// TIA Portal project "Wine Bottling" (V16)

(* hardware
DEVICE "S71500/ET200MP station_1"  S7-1500 station
   slot 0: "Rail_0"  Rack  6ES7 590-1***0-0AA0
   slot 1: "PLC_1"  CPU 1512C-1 PN  6ES7 512-1CK00-0AB0  V2.8
      slot 3: "CPU display_1"  6ES7591-1AA00-0AA0
      slot 32768: "PROFINET interface_1"  X1
         slot 32769: "Port_1"  X1 P1
         slot 32770: "Port_2"  X1 P2
      slot 34817: "Virtual CP interface port_1"  Virtual CP interface port  Virtual CP interface port
DEVICE "HMI_1"  TP1200 Comfort
   slot 0: "HMI_1"  TP1200 Comfort  6AV2 124-0MC01-0AX0  16.0.0.0
   slot 1: "HMI_RT_1"  TP1200 Comfort  6AV2 124-0MC01-0AX0  16.0.0.0
   slot 5: "HMI_1.IE_CP_1"  PROFINET Interface  16.0.0.0
      slot 1: "PROFINET Interface_1"  PROFINET Interface
         slot 1: "Port_1"  Port
         slot 2: "Port_2"  Port
   slot 7: "HMI_1.MPI/DP_CP_1"  MPI/DP Interface  16.0.0.0
*)

// ===== PLC "PLC_1"  CPU 1512C-1 PN =====

VAR_GLOBAL   // PLC tag table "Default tag table"
   "Start" AT %M0.0 : Bool;
   "Production line" AT %M0.1 : Bool;
   "P_TRIG" AT %M0.2 : Bool;
   "WhiteBottleSensor" AT %M0.3 : Bool;
   "DarkBottleSensor" AT %M0.4 : Bool;
   "Filling" AT %M0.5 : Bool;
   "P_TRIG1" AT %M0.6 : Bool;
   "FillingWhiteWine" AT %M0.7 : Bool;
   "FillingDarkWine" AT %M1.0 : Bool;
   "P_TRIG2" AT %M1.1 : Bool;
   "FilWhite" AT %M1.2 : Bool;
   "FillDark" AT %M1.3 : Bool;
   "P_TRIG3" AT %M1.4 : Bool;
   "P_TRIG4" AT %M1.5 : Bool;
   "P_TRIG5" AT %M1.6 : Bool;
   "Corking" AT %M1.7 : Bool;
   "CorkingWhite" AT %M2.0 : Bool;
   "CorkingDark" AT %M2.1 : Bool;
   "P_TRIG7" AT %M2.2 : Bool;
   "P_TRIG6" AT %M2.3 : Bool;
   "CorkingDarkWine" AT %M2.4 : Bool;
   "P_TRIG8" AT %M2.5 : Bool;
   "CorkingWhiteWine" AT %M2.6 : Bool;
   "P_TRIG9" AT %M2.7 : Bool;
   "P_TRIG10" AT %M3.0 : Bool;
   "Label" AT %M3.1 : Bool;
   "LabelWhite" AT %M3.2 : Bool;
   "LabelDark" AT %M3.3 : Bool;
   "P_TRIG13" AT %M3.4 : Bool;
   "P_TRIG14" AT %M3.5 : Bool;
   "P_TRIG11" AT %M3.6 : Bool;
   "P_TRIG12" AT %M3.7 : Bool;
   "LabelWhiteWine" AT %M4.0 : Bool;
   "LabelDarkWine" AT %M4.1 : Bool;
   "P_TRIG15" AT %M4.2 : Bool;
   "P_TRIG17" AT %M4.3 : Bool;
   "P_TRIG16" AT %M4.4 : Bool;
   "NeckLabeling" AT %M4.5 : Bool;
   "NeckLabelWhite" AT %M4.6 : Bool;
   "NeckLabelDark" AT %M4.7 : Bool;
   "P_TRIG19" AT %M5.0 : Bool;
   "P_TRIG18" AT %M5.1 : Bool;
   "NeckLabelWhiteWine" AT %M5.2 : Bool;
   "NeckLabelDarkWine" AT %M5.3 : Bool;
   "P_TRIG20" AT %M5.4 : Bool;
END_VAR

ORGANIZATION_BLOCK "Main"   // OB1, LAD, ProgramCycle
TITLE = "Main Program Sweep (Cycle)"
{ S7_Optimized_Access := 'TRUE' }
VERSION : 0.1
   VAR_INPUT
      Initial_Call : Bool;   // Initial call of this OB
      Remanence : Bool;   // =True, if remanent data are available
   END_VAR
   VAR_TEMP   // added for the SCL form of the ladder/FBD networks
      _w1 : Bool;
      _w2 : Bool;
      _w3 : Bool;
      _w4 : Bool;
   END_VAR
BEGIN

REGION Network 1
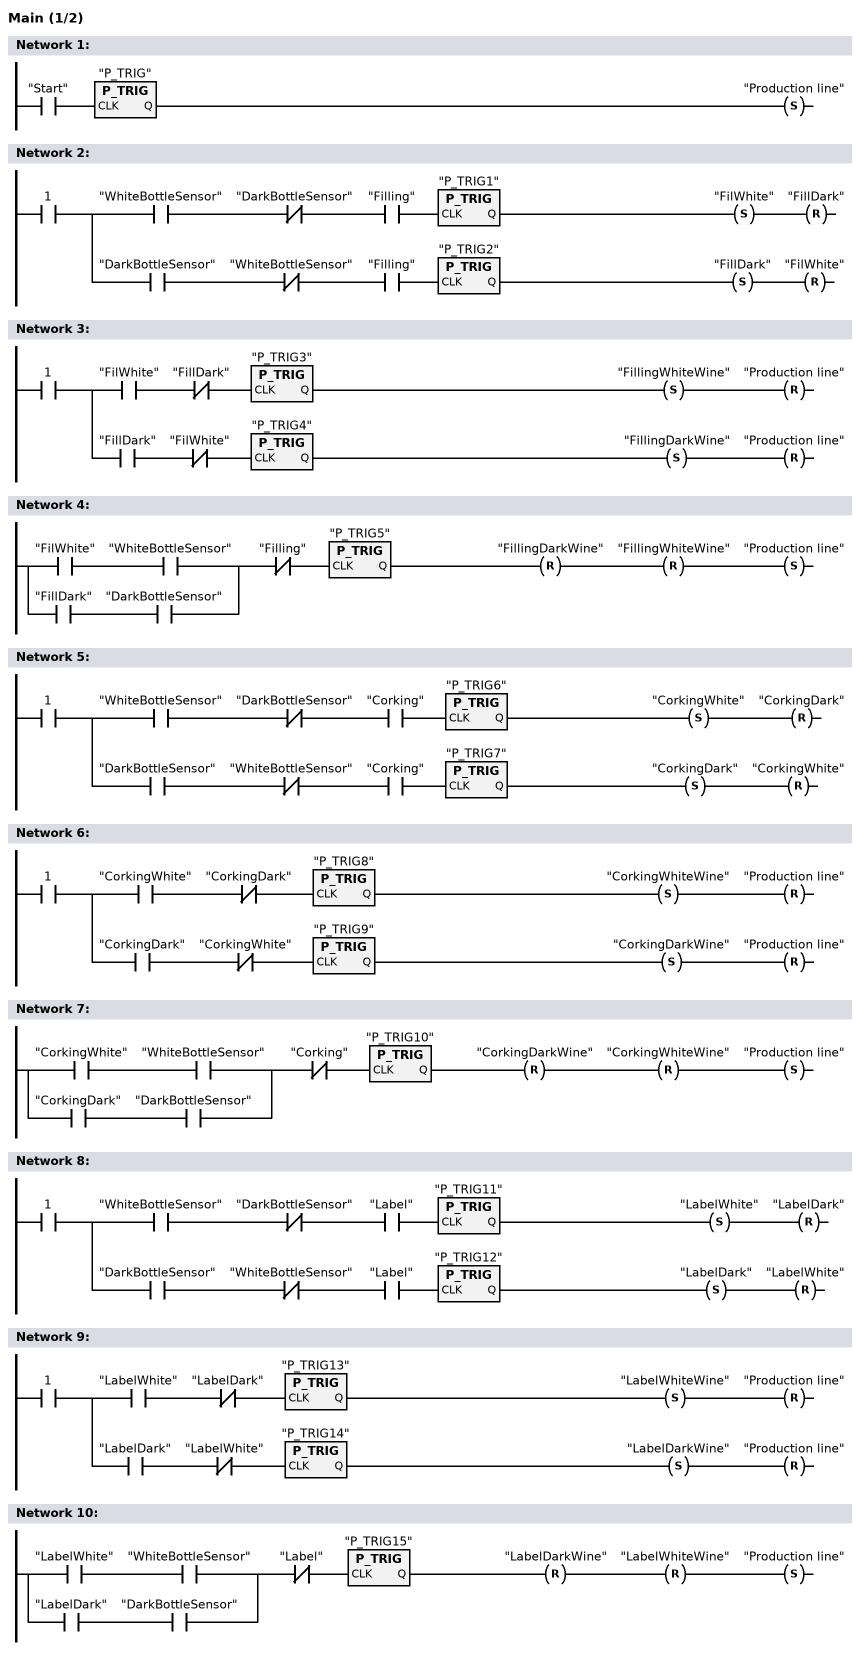
   RUNG wire#powerrail
      Contact( "Start" )
      P_Trig( "P_TRIG" )
      S_Coil( "Production line" )
   END_RUNG
   // the same network as SCL:
   #_w1 := "Start" AND NOT "P_TRIG";   // rising edge
   "P_TRIG" := "Start";
   IF #_w1 THEN "Production line" := TRUE; END_IF;
END_REGION

REGION Network 2
   RUNG wire#powerrail
      Contact( 1 )
      wire#w1
      Contact( "WhiteBottleSensor" )
      I_Contact( "DarkBottleSensor" )
      Contact( "Filling" )
      P_Trig( "P_TRIG1" )
      S_Coil( "FilWhite" )
      R_Coil( "FillDark" )
   END_RUNG
   RUNG wire#w1
      Contact( "DarkBottleSensor" )
      I_Contact( "WhiteBottleSensor" )
      Contact( "Filling" )
      P_Trig( "P_TRIG2" )
      S_Coil( "FillDark" )
      R_Coil( "FilWhite" )
   END_RUNG
   // the same network as SCL:
   #_w1 := 1 AND "WhiteBottleSensor" AND NOT "DarkBottleSensor" AND "Filling";
   #_w2 := #_w1 AND NOT "P_TRIG1";   // rising edge
   "P_TRIG1" := #_w1;
   IF #_w2 THEN
       "FilWhite" := TRUE;
       "FillDark" := FALSE;
   END_IF;
   #_w3 := 1 AND "DarkBottleSensor" AND NOT "WhiteBottleSensor" AND "Filling";
   #_w4 := #_w3 AND NOT "P_TRIG2";   // rising edge
   "P_TRIG2" := #_w3;
   IF #_w4 THEN
       "FillDark" := TRUE;
       "FilWhite" := FALSE;
   END_IF;
END_REGION

REGION Network 3
   RUNG wire#powerrail
      Contact( 1 )
      wire#w1
      Contact( "FilWhite" )
      I_Contact( "FillDark" )
      P_Trig( "P_TRIG3" )
      S_Coil( "FillingWhiteWine" )
      R_Coil( "Production line" )
   END_RUNG
   RUNG wire#w1
      Contact( "FillDark" )
      I_Contact( "FilWhite" )
      P_Trig( "P_TRIG4" )
      S_Coil( "FillingDarkWine" )
      R_Coil( "Production line" )
   END_RUNG
   // the same network as SCL:
   #_w1 := 1 AND "FilWhite" AND NOT "FillDark";
   #_w2 := #_w1 AND NOT "P_TRIG3";   // rising edge
   "P_TRIG3" := #_w1;
   IF #_w2 THEN
       "FillingWhiteWine" := TRUE;
       "Production line" := FALSE;
   END_IF;
   #_w3 := 1 AND "FillDark" AND NOT "FilWhite";
   #_w4 := #_w3 AND NOT "P_TRIG4";   // rising edge
   "P_TRIG4" := #_w3;
   IF #_w4 THEN
       "FillingDarkWine" := TRUE;
       "Production line" := FALSE;
   END_IF;
END_REGION

REGION Network 4
   RUNG wire#powerrail
      Contact( "FilWhite" )
      Contact( "WhiteBottleSensor" )
      wire#w1
      I_Contact( "Filling" )
      P_Trig( "P_TRIG5" )
      R_Coil( "FillingDarkWine" )
      R_Coil( "FillingWhiteWine" )
      S_Coil( "Production line" )
   END_RUNG
   RUNG wire#powerrail
      Contact( "FillDark" )
      Contact( "DarkBottleSensor" )
   END_RUNG wire#w1
   // the same network as SCL:
   #_w1 := (("FilWhite" AND "WhiteBottleSensor") OR ("FillDark" AND "DarkBottleSensor")) AND NOT "Filling";
   #_w2 := #_w1 AND NOT "P_TRIG5";   // rising edge
   "P_TRIG5" := #_w1;
   IF #_w2 THEN
       "FillingDarkWine" := FALSE;
       "FillingWhiteWine" := FALSE;
       "Production line" := TRUE;
   END_IF;
END_REGION

REGION Network 5
   RUNG wire#powerrail
      Contact( 1 )
      wire#w1
      Contact( "WhiteBottleSensor" )
      I_Contact( "DarkBottleSensor" )
      Contact( "Corking" )
      P_Trig( "P_TRIG6" )
      S_Coil( "CorkingWhite" )
      R_Coil( "CorkingDark" )
   END_RUNG
   RUNG wire#w1
      Contact( "DarkBottleSensor" )
      I_Contact( "WhiteBottleSensor" )
      Contact( "Corking" )
      P_Trig( "P_TRIG7" )
      S_Coil( "CorkingDark" )
      R_Coil( "CorkingWhite" )
   END_RUNG
   // the same network as SCL:
   #_w1 := 1 AND "WhiteBottleSensor" AND NOT "DarkBottleSensor" AND "Corking";
   #_w2 := #_w1 AND NOT "P_TRIG6";   // rising edge
   "P_TRIG6" := #_w1;
   IF #_w2 THEN
       "CorkingWhite" := TRUE;
       "CorkingDark" := FALSE;
   END_IF;
   #_w3 := 1 AND "DarkBottleSensor" AND NOT "WhiteBottleSensor" AND "Corking";
   #_w4 := #_w3 AND NOT "P_TRIG7";   // rising edge
   "P_TRIG7" := #_w3;
   IF #_w4 THEN
       "CorkingDark" := TRUE;
       "CorkingWhite" := FALSE;
   END_IF;
END_REGION

REGION Network 6
   RUNG wire#powerrail
      Contact( 1 )
      wire#w1
      Contact( "CorkingWhite" )
      I_Contact( "CorkingDark" )
      P_Trig( "P_TRIG8" )
      S_Coil( "CorkingWhiteWine" )
      R_Coil( "Production line" )
   END_RUNG
   RUNG wire#w1
      Contact( "CorkingDark" )
      I_Contact( "CorkingWhite" )
      P_Trig( "P_TRIG9" )
      S_Coil( "CorkingDarkWine" )
      R_Coil( "Production line" )
   END_RUNG
   // the same network as SCL:
   #_w1 := 1 AND "CorkingWhite" AND NOT "CorkingDark";
   #_w2 := #_w1 AND NOT "P_TRIG8";   // rising edge
   "P_TRIG8" := #_w1;
   IF #_w2 THEN
       "CorkingWhiteWine" := TRUE;
       "Production line" := FALSE;
   END_IF;
   #_w3 := 1 AND "CorkingDark" AND NOT "CorkingWhite";
   #_w4 := #_w3 AND NOT "P_TRIG9";   // rising edge
   "P_TRIG9" := #_w3;
   IF #_w4 THEN
       "CorkingDarkWine" := TRUE;
       "Production line" := FALSE;
   END_IF;
END_REGION

REGION Network 7
   RUNG wire#powerrail
      Contact( "CorkingWhite" )
      Contact( "WhiteBottleSensor" )
      wire#w1
      I_Contact( "Corking" )
      P_Trig( "P_TRIG10" )
      R_Coil( "CorkingDarkWine" )
      R_Coil( "CorkingWhiteWine" )
      S_Coil( "Production line" )
   END_RUNG
   RUNG wire#powerrail
      Contact( "CorkingDark" )
      Contact( "DarkBottleSensor" )
   END_RUNG wire#w1
   // the same network as SCL:
   #_w1 := (("CorkingWhite" AND "WhiteBottleSensor") OR ("CorkingDark" AND "DarkBottleSensor")) AND NOT "Corking";
   #_w2 := #_w1 AND NOT "P_TRIG10";   // rising edge
   "P_TRIG10" := #_w1;
   IF #_w2 THEN
       "CorkingDarkWine" := FALSE;
       "CorkingWhiteWine" := FALSE;
       "Production line" := TRUE;
   END_IF;
END_REGION

REGION Network 8
   RUNG wire#powerrail
      Contact( 1 )
      wire#w1
      Contact( "WhiteBottleSensor" )
      I_Contact( "DarkBottleSensor" )
      Contact( "Label" )
      P_Trig( "P_TRIG11" )
      S_Coil( "LabelWhite" )
      R_Coil( "LabelDark" )
   END_RUNG
   RUNG wire#w1
      Contact( "DarkBottleSensor" )
      I_Contact( "WhiteBottleSensor" )
      Contact( "Label" )
      P_Trig( "P_TRIG12" )
      S_Coil( "LabelDark" )
      R_Coil( "LabelWhite" )
   END_RUNG
   // the same network as SCL:
   #_w1 := 1 AND "WhiteBottleSensor" AND NOT "DarkBottleSensor" AND "Label";
   #_w2 := #_w1 AND NOT "P_TRIG11";   // rising edge
   "P_TRIG11" := #_w1;
   IF #_w2 THEN
       "LabelWhite" := TRUE;
       "LabelDark" := FALSE;
   END_IF;
   #_w3 := 1 AND "DarkBottleSensor" AND NOT "WhiteBottleSensor" AND "Label";
   #_w4 := #_w3 AND NOT "P_TRIG12";   // rising edge
   "P_TRIG12" := #_w3;
   IF #_w4 THEN
       "LabelDark" := TRUE;
       "LabelWhite" := FALSE;
   END_IF;
END_REGION

REGION Network 9
   RUNG wire#powerrail
      Contact( 1 )
      wire#w1
      Contact( "LabelWhite" )
      I_Contact( "LabelDark" )
      P_Trig( "P_TRIG13" )
      S_Coil( "LabelWhiteWine" )
      R_Coil( "Production line" )
   END_RUNG
   RUNG wire#w1
      Contact( "LabelDark" )
      I_Contact( "LabelWhite" )
      P_Trig( "P_TRIG14" )
      S_Coil( "LabelDarkWine" )
      R_Coil( "Production line" )
   END_RUNG
   // the same network as SCL:
   #_w1 := 1 AND "LabelWhite" AND NOT "LabelDark";
   #_w2 := #_w1 AND NOT "P_TRIG13";   // rising edge
   "P_TRIG13" := #_w1;
   IF #_w2 THEN
       "LabelWhiteWine" := TRUE;
       "Production line" := FALSE;
   END_IF;
   #_w3 := 1 AND "LabelDark" AND NOT "LabelWhite";
   #_w4 := #_w3 AND NOT "P_TRIG14";   // rising edge
   "P_TRIG14" := #_w3;
   IF #_w4 THEN
       "LabelDarkWine" := TRUE;
       "Production line" := FALSE;
   END_IF;
END_REGION

REGION Network 10
   RUNG wire#powerrail
      Contact( "LabelWhite" )
      Contact( "WhiteBottleSensor" )
      wire#w1
      I_Contact( "Label" )
      P_Trig( "P_TRIG15" )
      R_Coil( "LabelDarkWine" )
      R_Coil( "LabelWhiteWine" )
      S_Coil( "Production line" )
   END_RUNG
   RUNG wire#powerrail
      Contact( "LabelDark" )
      Contact( "DarkBottleSensor" )
   END_RUNG wire#w1
   // the same network as SCL:
   #_w1 := (("LabelWhite" AND "WhiteBottleSensor") OR ("LabelDark" AND "DarkBottleSensor")) AND NOT "Label";
   #_w2 := #_w1 AND NOT "P_TRIG15";   // rising edge
   "P_TRIG15" := #_w1;
   IF #_w2 THEN
       "LabelDarkWine" := FALSE;
       "LabelWhiteWine" := FALSE;
       "Production line" := TRUE;
   END_IF;
END_REGION

REGION Network 11
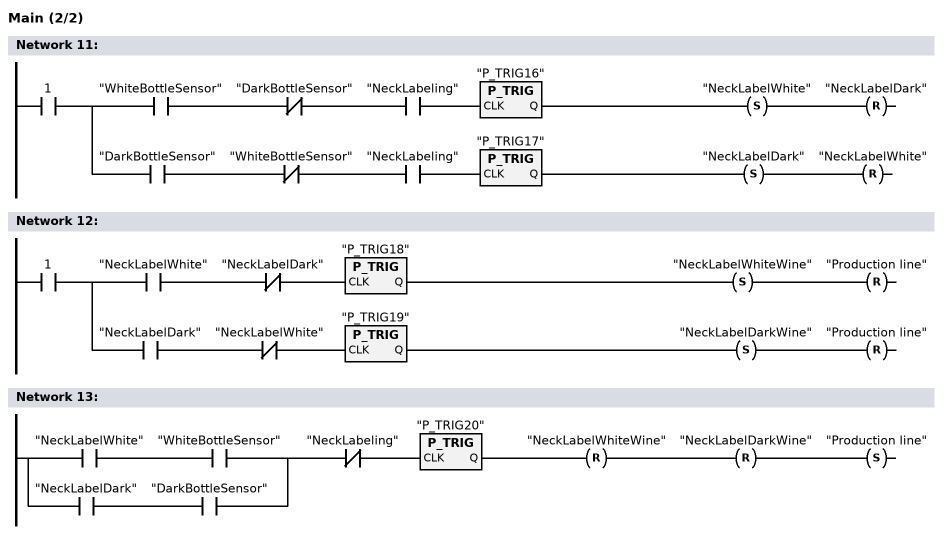
   RUNG wire#powerrail
      Contact( 1 )
      wire#w1
      Contact( "WhiteBottleSensor" )
      I_Contact( "DarkBottleSensor" )
      Contact( "NeckLabeling" )
      P_Trig( "P_TRIG16" )
      S_Coil( "NeckLabelWhite" )
      R_Coil( "NeckLabelDark" )
   END_RUNG
   RUNG wire#w1
      Contact( "DarkBottleSensor" )
      I_Contact( "WhiteBottleSensor" )
      Contact( "NeckLabeling" )
      P_Trig( "P_TRIG17" )
      S_Coil( "NeckLabelDark" )
      R_Coil( "NeckLabelWhite" )
   END_RUNG
   // the same network as SCL:
   #_w1 := 1 AND "WhiteBottleSensor" AND NOT "DarkBottleSensor" AND "NeckLabeling";
   #_w2 := #_w1 AND NOT "P_TRIG16";   // rising edge
   "P_TRIG16" := #_w1;
   IF #_w2 THEN
       "NeckLabelWhite" := TRUE;
       "NeckLabelDark" := FALSE;
   END_IF;
   #_w3 := 1 AND "DarkBottleSensor" AND NOT "WhiteBottleSensor" AND "NeckLabeling";
   #_w4 := #_w3 AND NOT "P_TRIG17";   // rising edge
   "P_TRIG17" := #_w3;
   IF #_w4 THEN
       "NeckLabelDark" := TRUE;
       "NeckLabelWhite" := FALSE;
   END_IF;
END_REGION

REGION Network 12
   RUNG wire#powerrail
      Contact( 1 )
      wire#w1
      Contact( "NeckLabelWhite" )
      I_Contact( "NeckLabelDark" )
      P_Trig( "P_TRIG18" )
      S_Coil( "NeckLabelWhiteWine" )
      R_Coil( "Production line" )
   END_RUNG
   RUNG wire#w1
      Contact( "NeckLabelDark" )
      I_Contact( "NeckLabelWhite" )
      P_Trig( "P_TRIG19" )
      S_Coil( "NeckLabelDarkWine" )
      R_Coil( "Production line" )
   END_RUNG
   // the same network as SCL:
   #_w1 := 1 AND "NeckLabelWhite" AND NOT "NeckLabelDark";
   #_w2 := #_w1 AND NOT "P_TRIG18";   // rising edge
   "P_TRIG18" := #_w1;
   IF #_w2 THEN
       "NeckLabelWhiteWine" := TRUE;
       "Production line" := FALSE;
   END_IF;
   #_w3 := 1 AND "NeckLabelDark" AND NOT "NeckLabelWhite";
   #_w4 := #_w3 AND NOT "P_TRIG19";   // rising edge
   "P_TRIG19" := #_w3;
   IF #_w4 THEN
       "NeckLabelDarkWine" := TRUE;
       "Production line" := FALSE;
   END_IF;
END_REGION

REGION Network 13
   RUNG wire#powerrail
      Contact( "NeckLabelWhite" )
      Contact( "WhiteBottleSensor" )
      wire#w1
      I_Contact( "NeckLabeling" )
      P_Trig( "P_TRIG20" )
      R_Coil( "NeckLabelWhiteWine" )
      R_Coil( "NeckLabelDarkWine" )
      S_Coil( "Production line" )
   END_RUNG
   RUNG wire#powerrail
      Contact( "NeckLabelDark" )
      Contact( "DarkBottleSensor" )
   END_RUNG wire#w1
   // the same network as SCL:
   #_w1 := (("NeckLabelWhite" AND "WhiteBottleSensor") OR ("NeckLabelDark" AND "DarkBottleSensor")) AND NOT "NeckLabeling";
   #_w2 := #_w1 AND NOT "P_TRIG20";   // rising edge
   "P_TRIG20" := #_w1;
   IF #_w2 THEN
       "NeckLabelWhiteWine" := FALSE;
       "NeckLabelDarkWine" := FALSE;
       "Production line" := TRUE;
   END_IF;
END_REGION
END_ORGANIZATION_BLOCK

(* ===== HMI "HMI_RT_1" =====
system functions are stored by id; their names below are inferred from use
connection "HMI_Connection_1": ETHERNET, S7_1500_OMS

HMI tags "Default tag table"
   "Tag_ScreenNumber" : UInt, internal
   "Start" : Bool = PLC Start AT %M0.0, 1 s
   "Production line" : Bool = PLC "Production line" AT %M0.1, 1 s
   "WhiteBottleSensor" : Bool = PLC WhiteBottleSensor AT %M0.3, 1 s
   "Filling" : Bool = PLC Filling AT %M0.5, 1 s
   "FillingWhiteWine" : Bool = PLC FillingWhiteWine AT %M0.7, 1 s
   "DarkBottleSensor" : Bool = PLC DarkBottleSensor AT %M0.4, 1 s
   "FillingDarkWine" : Bool = PLC FillingDarkWine AT %M1.0, 1 s
   "Corking" : Bool = PLC Corking AT %M1.7, 1 s
   "CorkingWhiteWine" : Bool = PLC CorkingWhiteWine AT %M2.6, 1 s
   "CorkingDarkWine" : Bool = PLC CorkingDarkWine AT %M2.4, 1 s
   "Label" : Bool = PLC Label AT %M3.1, 1 s
   "LabelWhiteWine" : Bool = PLC LabelWhiteWine AT %M4.0, 1 s
   "LabelDarkWine" : Bool = PLC LabelDarkWine AT %M4.1, 1 s
   "NeckLabeling" : Bool = PLC NeckLabeling AT %M4.5, 1 s
   "NeckLabelWhiteWine" : Bool = PLC NeckLabelWhiteWine AT %M5.2, 1 s
   "NeckLabelDarkWine" : Bool = PLC NeckLabelDarkWine AT %M5.3, 1 s

screen "Root screen" 1280x740, template "Template_1"
   on GenerateScreen: SetTag("Tag_ScreenNumber", 1)
   Button "Button_1" at 103,77 size 96x32; TextOff 'Start'
      on Press: InvertBit("Start")
   Circle "Circle_1" at 257,67 size 48x48
      Appearance <- "Start"
   TextField "Text field_1" at 53,142 size 155x25; Text 'Production Line'
   Circle "Circle_2" at 257,124 size 48x48
      Appearance <- "Production line"
   Button "Button_2" at 55,190 size 179x32; TextOff 'White Bottle Sensor'
      on Press: InvertBit("WhiteBottleSensor")
   Circle "Circle_3" at 258,180 size 48x48
      Appearance <- "WhiteBottleSensor"
   Button "Button_4" at 61,250 size 96x32; TextOff 'Filling'
      on Press: InvertBit("Filling")
   Circle "Circle_5" at 258,239 size 48x48
      Appearance <- "Filling"
   TextField "Text field_2" at 443,77 size 148x25; Text 'Fill White Wine'
   Circle "Circle_6" at 612,46 size 48x48
      Appearance <- "FillingWhiteWine"
   Button "Button_3" at 61,313 size 179x32; TextOff 'Dark Bottle Sensor'
      on Press: InvertBit("DarkBottleSensor")
   Circle "Circle_4" at 258,305 size 48x48
      Appearance <- "DarkBottleSensor"
   TextField "Text field_3" at 448,127 size 137x25; Text 'Fill Dark Wine'
   Circle "Circle_7" at 618,113 size 48x48
      Appearance <- "FillingDarkWine"
   TextField "Text field_4" at 443,309 size 17x25; Text 'Text'
   Button "Button_5" at 69,376 size 96x32; TextOff 'Corking'
      on Press: InvertBit("Corking")
   Circle "Circle_8" at 257,366 size 48x48
      Appearance <- "Corking"
   Circle "Circle_9" at 618,191 size 48x48
      Appearance <- "CorkingWhiteWine"
   Circle "Circle_10" at 618,256 size 48x48
      Appearance <- "CorkingDarkWine"
   TextField "Text field_5" at 420,201 size 192x25; Text 'Corking White Wine'
   TextField "Text field_6" at 431,274 size 181x25; Text 'Corking Dark Wine'
   Button "Button_6" at 70,453 size 96x32; TextOff 'Label'
      on Press: InvertBit("Label")
   Circle "Circle_11" at 257,443 size 48x48
      Appearance <- "Label"
   TextField "Text field_7" at 431,332 size 170x25; Text 'Label White Wine'
   TextField "Text field_8" at 431,395 size 159x25; Text 'Label Dark Wine'
   Circle "Circle_12" at 621,318 size 48x48
      Appearance <- "LabelWhiteWine"
   Circle "Circle_13" at 621,380 size 48x48
      Appearance <- "LabelDarkWine"
   Button "Button_7" at 61,523 size 110x32; TextOff 'Neck Label'
      on Press: InvertBit("NeckLabeling")
   Circle "Circle_14" at 258,508 size 48x48
      Appearance <- "NeckLabeling"
   TextField "Text field_9" at 430,460 size 175x25; Text 'Neck Label White'
   Circle "Circle_15" at 621,440 size 48x48
      Appearance <- "NeckLabelWhiteWine"
   TextField "Text field_10" at 431,506 size 158x25; Text 'Neck Label Dark'
   Circle "Circle_16" at 621,491 size 48x48
      Appearance <- "NeckLabelDarkWine"

Template "Template_1" 1280x740
   Button "Exit" at 1200,679 size 78x59; TextOff 'Exit'; PictureOff "ExitRuntime_TP1200_Comfort_TR"; PictureOn "ExitRuntime_TP1200_Comfort_TR"
      on Release: StopRuntime(0)
   Button "Template_Button" at 1120,679 size 78x59; TextOff 'Text'
   Button "Template_Button_1" at 1040,679 size 78x59; TextOff 'Text'
   Button "Template_Button_2" at 960,679 size 78x59; TextOff 'Text'
   Button "Template_Button_3" at 880,679 size 78x59; TextOff 'Text'
   Button "Template_Button_4" at 800,679 size 78x59; TextOff 'Text'
   Button "Template_Button_5" at 720,679 size 78x59; TextOff 'Text'
   Button "Template_Button_6" at 640,679 size 78x59; TextOff 'Text'
   Button "Template_Button_7" at 561,679 size 78x59; TextOff 'Text'
   Button "Template_Button_8" at 481,679 size 78x59; TextOff 'Text'
   Button "Template_Button_9" at 401,679 size 78x59; TextOff 'Text'
   Button "Template_Button_10" at 321,679 size 78x59; TextOff 'Text'
   Button "Template_Button_11" at 241,679 size 78x59; TextOff 'Text'
   Button "Template_Button_12" at 161,679 size 78x59; TextOff 'Text'
   Button "Template_Button_13" at 81,679 size 78x59; TextOff 'Text'
   Button "Start screen" at 1,679 size 78x59; TextOff 'Start screen'; PictureOff "NavigateHome_TP1200_Comfort_TR"; PictureOn "NavigateHome_TP1200_Comfort_TR"
      on Release: ActivateScreen("Root screen", 0)
*)